(* PLC project Generated.project, CODESYS CODESYS V3.5 SP19 Patch 1 *)
(* stored: creationDateTime 2026-09-01T00:57:57.847775, modificationDateTime 2026-09-01T00:57:57.847775 *)

(* ═══════════════════════════════════════════════════════════════ 🚦 ST_CycleExtractionState — États publics cycle extraction ═══════════════════════════════════════════════════════════════ *)
TYPE ST_CycleExtractionState : STRUCT
  ExtractionReady : BOOL;
  ExtractionBusy : BOOL;
  ExtractionDone : BOOL;
  ExtractionError : BOOL;
  ExtractionErrorId : WORD;
  ExtractionState : E_ExtractionAssistState;
  ExtractionStepAtFault : E_ExtractionAssistState;
END_STRUCT;
END_TYPE
